// TIA Portal project "babu_risingEdge" (V15)

(* hardware
DEVICE "S7-1200 station_1"  S7-1200 Station
   slot 0: "Rack_0"  S7-1200 Rack  Rack  V1.0
   slot 1: "PLC_1"  CPU 1212C DC/DC/DC  6ES7 212-1AE40-0XB0  V4.2
*)

// ===== PLC "PLC_1"  CPU 1212C DC/DC/DC =====

VAR_GLOBAL   // PLC tag table "Default tag table"
   "INPUT" AT %M0.0 : Bool;
   "OUTPUT" AT %Q0.0 : Bool;
   "IP1" AT %M0.1 : Bool;
   "NA1" AT %M0.2 : Bool;
   "OP1" AT %Q0.1 : Bool;
   "IP2" AT %M0.3 : Bool;
   "OP2" AT %M0.4 : Bool;
   "MEM2" AT %M0.5 : Bool;
   "IP3" AT %M0.6 : Bool;
   "OP3" AT %M0.7 : Bool;
   "MEM3" AT %M1.0 : Bool;
   "OP5" AT %M1.1 : Bool;
   "MEM5" AT %M1.2 : Bool;
   "MEM51" AT %M1.3 : Bool;
   "OP51" AT %Q0.2 : Bool;
   "IP6" AT %M1.4 : Bool;
   "MEM61" AT %M1.5 : Bool;
   "MEM62" AT %M1.6 : Bool;
   "OP6" AT %Q0.3 : Bool;
END_VAR

ORGANIZATION_BLOCK "Main"   // OB1, LAD, ProgramCycle
TITLE = "Main Program Sweep (Cycle)"
{ S7_Optimized_Access := 'TRUE' }
VERSION : 0.1
   VAR_INPUT
      Initial_Call : Bool;   // Initial call of this OB
      Remanence : Bool;   // =True, if remanent data are available
   END_VAR
   VAR_TEMP   // added for the SCL form of the ladder/FBD networks
      _w1 : Bool;
   END_VAR
BEGIN

REGION Network 1
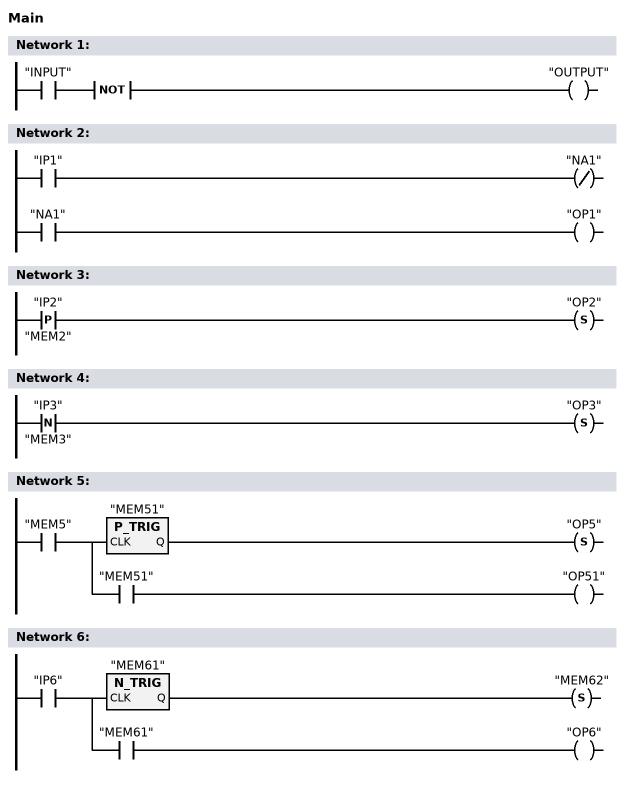
   RUNG wire#powerrail
      Contact( "INPUT" )
      Not()
      Coil( "OUTPUT" )
   END_RUNG
   // the same network as SCL:
   "OUTPUT" := NOT "INPUT";
END_REGION

REGION Network 2
   RUNG wire#powerrail
      Contact( "IP1" )
      I_Coil( "NA1" )
   END_RUNG
   RUNG wire#powerrail
      Contact( "NA1" )
      Coil( "OP1" )
   END_RUNG
   // the same network as SCL:
   "NA1" := NOT "IP1";
   "OP1" := "NA1";
END_REGION

REGION Network 3
   RUNG wire#powerrail
      P_Contact(operand := "IP2", bit := "MEM2")
      S_Coil( "OP2" )
   END_RUNG
   // the same network as SCL:
   #_w1 := "IP2" AND NOT "MEM2";   // rising edge of "IP2"
   "MEM2" := "IP2";
   IF #_w1 THEN "OP2" := TRUE; END_IF;
END_REGION

REGION Network 4
   RUNG wire#powerrail
      N_Contact(operand := "IP3", bit := "MEM3")
      S_Coil( "OP3" )
   END_RUNG
   // the same network as SCL:
   #_w1 := NOT "IP3" AND "MEM3";   // falling edge of "IP3"
   "MEM3" := "IP3";
   IF #_w1 THEN "OP3" := TRUE; END_IF;
END_REGION

REGION Network 5
   RUNG wire#powerrail
      Contact( "MEM5" )
      wire#w1
      P_Trig( "MEM51" )
      S_Coil( "OP5" )
   END_RUNG
   RUNG wire#w1
      Contact( "MEM51" )
      Coil( "OP51" )
   END_RUNG
   // the same network as SCL:
   #_w1 := "MEM5" AND NOT "MEM51";   // rising edge
   "MEM51" := "MEM5";
   IF #_w1 THEN "OP5" := TRUE; END_IF;
   "OP51" := "MEM5" AND "MEM51";
END_REGION

REGION Network 6
   RUNG wire#powerrail
      Contact( "IP6" )
      wire#w1
      N_Trig( "MEM61" )
      S_Coil( "MEM62" )
   END_RUNG
   RUNG wire#w1
      Contact( "MEM61" )
      Coil( "OP6" )
   END_RUNG
   // the same network as SCL:
   #_w1 := NOT "IP6" AND "MEM61";   // falling edge
   "MEM61" := "IP6";
   IF #_w1 THEN "MEM62" := TRUE; END_IF;
   "OP6" := "IP6" AND "MEM61";
END_REGION
END_ORGANIZATION_BLOCK